// TIA Portal V20 export
// export: Created 2026-04-11T06:02:30.1619486Z, ExportSetting WithDefaults, DisplayName Totally Integrated Automation Portal, DisplayVersion V20, DisplayName TIA Portal Openness, DisplayVersion V20, DisplayName TIA Portal Version Control Interface, DisplayVersion V20, DisplayName STEP 7 Professional, DisplayVersion V20, DisplayName STEP 7 Safety, DisplayVersion V20, DisplayName WinCC Basic/Comfort/Advanced, DisplayVersion V20, DisplayName WinCC Unified, DisplayVersion V20
TYPE "udtHMI_MotorControl"
// stored: IsFailsafeCompliant false
   STRUCT
      iMode : Int;   // Current mode
      iErrorCode { ExternalWritable := 'False'} : Int;   // Error code
      iStatus { ExternalWritable := 'False'} : Int;   // Status for HMI display
      bPB_ResetError : Bool;   // PB Reset block errors
      bPB_Forward : Bool;   // PB Move forward in manual mode
      bPB_Reverse : Bool;   // PB Move Reverse in manual mode
      bPB_Stop : Bool;   // PB Stop in manual mode
      bPBEN_ResetError { ExternalWritable := 'False'} : Bool;   // PB Reset error enabled
      bPBEN_Forward { ExternalWritable := 'False'} : Bool;   // PB Forward enabled
      bPBEN_Reverse { ExternalWritable := 'False'} : Bool;   // PB Reverse enabled
      bPBEN_Stop { ExternalWritable := 'False'} : Bool;   // PB Stop enabled
      bForwardOn { ExternalWritable := 'False'} : Bool;   // Moving forward
      bReverseOn { ExternalWritable := 'False'} : Bool;   // Moving Reverse
      bSignalForward { ExternalWritable := 'False'} : Bool;   // Forward signal
      bSignalReverse { ExternalWritable := 'False'} : Bool;   // Reverse signal
      bError { ExternalWritable := 'False'} : Bool;   // Overall error
      bInterlock { ExternalWritable := 'False'} : Bool;   // Motor interlocked
   END_STRUCT;
END_TYPE
